SYSTEM System (* System Configuration *)
  (* Standard: 61499-1 *)
  (* Version 0.0, 9/26/2014, cheyan, nxtControl GmbH *)
  {SET_ATTRIBUTE(System.Device.FolderPath, DEV1,DEV2)}
  APPLICATION APP1
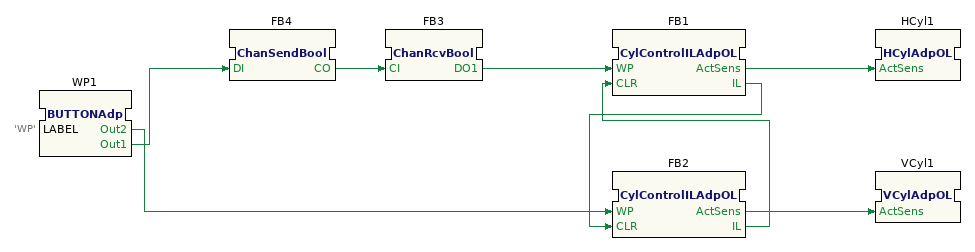
    FBS
      HCyl1 : HCylAdpOL;
      VCyl1 : VCylAdpOL;
      WP1 : BUTTONAdp(LABEL := 'WP');
      FB1 : CylControlILAdpOL;
      FB2 : CylControlILAdpOL;
      FB3 : ChanRcvBool;
      FB4 : ChanSendBool;
    END_FBS
    ADAPTER_CONNECTIONS
      FB1.ActSens TO HCyl1.ActSens;
      FB2.ActSens TO VCyl1.ActSens;
      FB3.DO1 TO FB1.WP;
      WP1.Out2 TO FB2.WP;
      FB4.CO TO FB3.CI;
      WP1.Out1 TO FB4.DI;
      FB1.IL TO FB2.CLR;
      FB2.IL TO FB1.CLR;
    END_CONNECTIONS
  END_APPLICATION
  APPLICATION APP2
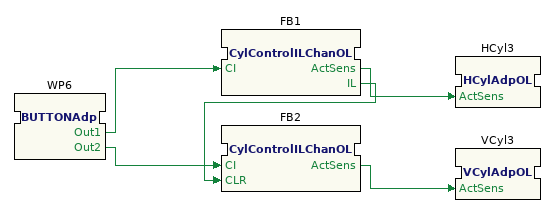
    FBS
      HCyl3 : HCylAdpOL;
      VCyl3 : VCylAdpOL;
      WP6 : BUTTONAdp;
      FB1 : CylControlILChanOL;
      FB2 : CylControlILChanOL;
    END_FBS
    ADAPTER_CONNECTIONS
      WP6.Out1 TO FB1.CI;
      WP6.Out2 TO FB2.CI;
      FB1.ActSens TO HCyl3.ActSens;
      FB1.IL TO FB2.CLR;
      FB2.ActSens TO VCyl3.ActSens;
    END_CONNECTIONS
  END_APPLICATION
  DEVICE DEV1 : Soft_dPAC
    RESOURCE RES0 : EMB_RES_ECO
      FBS
        WP1 : BUTTONAdp(LABEL := 'WP');
        FB4 : ChanSendBool;
        HCyl1 : HCylAdpOL;
        VCyl1 : VCylAdpOL;
        FB1 : CylControlILAdpOL;
        FB2 : CylControlILAdpOL;
        FB3 : ChanRcvBool;
        HCyl3 : HCylAdpOL;
        VCyl3 : VCylAdpOL;
      END_FBS
      ADAPTER_CONNECTIONS
        FB1.ActSens TO HCyl1.ActSens;
        FB2.ActSens TO VCyl1.ActSens;
        FB3.DO1 TO FB1.WP;
        WP1.Out2 TO FB2.WP;
        FB4.CO TO FB3.CI;
        WP1.Out1 TO FB4.DI;
        FB1.IL TO FB2.CLR;
        FB2.IL TO FB1.CLR;
      END_CONNECTIONS
    END_RESOURCE
  END_DEVICE
  DEVICE DEV2 : Soft_dPAC
    RESOURCE RES0 : EMB_RES_ECO
    END_RESOURCE
  END_DEVICE
  MAPPINGS
    APP1.WP1 ON DEV1.RES0;
    APP1.FB4 ON DEV1.RES0;
    APP1.HCyl1 ON DEV1.RES0;
    APP1.VCyl1 ON DEV1.RES0;
    APP1.FB1 ON DEV1.RES0;
    APP1.FB2 ON DEV1.RES0;
    APP1.FB3 ON DEV1.RES0;
    APP2.HCyl3 ON DEV1.RES0;
    APP2.VCyl3 ON DEV1.RES0;
  END_MAPPINGS
  SEGMENTS
    SEGMENT1 : localhost;
  END_SEGMENTS
END_SYSTEM
